FUNCTION_BLOCK TrafficLights
VAR_INPUT
END_VAR
VAR_OUTPUT
END_VAR
VAR
END_VAR

//This is where all the stuff you guys are going to add will go.

END_FUNCTION_BLOCK

(* stored: Version 1.1.0.1, ProductVersion 3.1.4024.11
   POU TrafficLights: Id {592c1bb7-9719-48f6-afbd-8153c16e6516}, SpecialFunc None *)
